// TIA Portal V17 export
// export: Created 2021-11-24T09:07:31.6775654Z, ExportSetting WithDefaults, DisplayName Totally Integrated Automation Portal, DisplayVersion V17, DisplayName TIA Portal Openness, DisplayVersion V17, DisplayName TIA Portal Version Control Interface, DisplayVersion V17, DisplayName SINAMICS Startdrive Advanced, DisplayVersion V17, DisplayName SINAMICS Startdrive G130, G150, S120, S150, SINAMICS MV, S210, DisplayVersion V17, DisplayName SINAMICS Startdrive G110M, G120, G120C, G120D, G120P, G115D, DisplayVersion V17, DisplayName STEP 7 Professional, DisplayVersion V17, DisplayName STEP 7 Safety, DisplayVersion V17, DisplayName WinCC Advanced / Unified PC, DisplayVersion V17
ORGANIZATION_BLOCK "SYNC_1"   // OB61, LAD, SynchronousCycle
TITLE = "DP Synchronous Interrupt"
VERSION : 0.1
// stored: IsIECCheckEnabled false
   VAR_TEMP
      OB61_EV_CLASS : Byte;   // Bits 0-3 = 1 (Coming event), Bits 4-7 = 1 (Event class 1)
      OB61_STRT_INF : Byte;   // OB 61 has started
      OB61_PRIORITY : Byte;   // Priority of OB Execution
      OB61_OB_NUMBR : Byte;   // 61 (Organization block 61, OB61)
      OB61_RESERVED_1 : Byte;   // Reserved for system
      OB61_RESERVED_2 : Byte;   // Reserved for system
      OB61_GC_VIOL : Bool;   // Lost Global Control of DP system
      OB61_FIRST : Bool;   // First Execution after startup or HALT
      OB61_MISSED_EXEC : Byte;   // Count of missed executions of OB61 since it was last scheduled
      OB61_DP_ID : Byte;   // DP master system ID of the synchronous DP system
      OB61_RESERVED_3 : Byte;   // Reserved for system
      OB61_RESERVED_4 : Word;   // Reserved for system
      OB61_DATE_TIME : Date_And_Time;   // Date and time OB61 started
   END_VAR
BEGIN

REGION Network 1
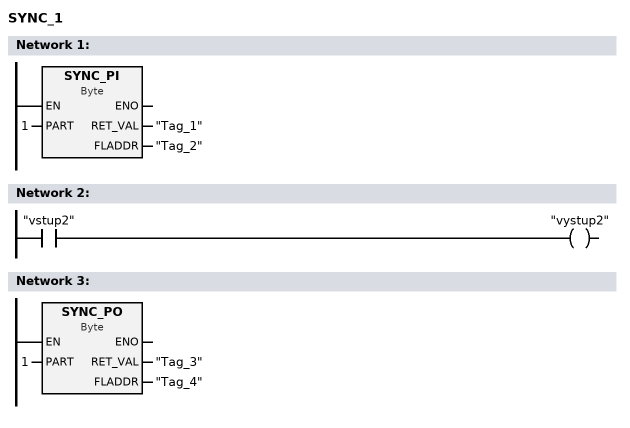
   RUNG wire#powerrail
      { S7_Templates := "value_type := Byte" } SYNC_PI(PART := 1, RET_VAL => "Tag_1", FLADDR => "Tag_2")
   END_RUNG
   // the same network as SCL:
   "Tag_1" := SYNC_PI(PART := 1, FLADDR => "Tag_2");
END_REGION

REGION Network 2
   RUNG wire#powerrail
      Contact( "vstup2" )
      Coil( "vystup2" )
   END_RUNG
   // the same network as SCL:
   "vystup2" := "vstup2";
END_REGION

REGION Network 3
   RUNG wire#powerrail
      { S7_Templates := "value_type := Byte" } SYNC_PO(PART := 1, RET_VAL => "Tag_3", FLADDR => "Tag_4")
   END_RUNG
   // the same network as SCL:
   "Tag_3" := SYNC_PO(PART := 1, FLADDR => "Tag_4");
END_REGION
END_ORGANIZATION_BLOCK
